FUNCTION_BLOCK FB_Roboter_Logik
VAR_INPUT
END_VAR
VAR_OUTPUT
END_VAR
VAR
END_VAR

END_FUNCTION_BLOCK

(* stored: Version 1.1.0.1, ProductVersion 3.1.4024.15
   POU FB_Roboter_Logik: Id {8ba7399c-3ab9-4824-9167-bb4531069ea3}, SpecialFunc None *)
